// THIS SHOULD BE COPIED AND NOT EXTENDED!!!
FUNCTION_BLOCK ABSTRACT AbstractRoom IMPLEMENTS I_Execute
VAR CONSTANT
	STATE_CAP		: UDINT := 4;
END_VAR
VAR
	_this			: Entity;
	_ctx			: Room_Ctx;
	_room			: RoomInterface(_ctx);
	_tag			: Tag(CONCAT('Room_', UDINT_TO_STRING(_room.Id)));
	_compTag		: Comp(_tag, _this);
	_exe			: Execute(THIS^);
	
	_uiLogic		: Room_UiLogic(_ctx);
	
	_onSystemEvent	: Room_OnSystemEvent(_ctx);
	
	_smgr			: StateManager<STATE_CAP>(_this);
	_proxSmgr		: StateManagerProxy(_smgr, _ctx.state.iMgr);
	
	_disable		: Room_State_Disabled(_this, _ctx);
	_proxDisable	: StateProxy(_disable, _ctx.state.iDisable);
	
	_fault			: Room_State_Fault(_this,_ctx);
	_proxFault		: StateProxy(_fault, _ctx.state.iFault);	
	
	_idle			: Room_State_Idle(_this,_ctx);
	_proxIdle		: StateProxy(_idle, _ctx.state.iIdle);	
	
	_systemOff		: Room_State_SystemOff(_this,_ctx);
	_proxSystemOff	: StateProxy(_systemOff, _ctx.state.iSystemOff);
END_VAR

	// Here add custom components

METHOD Execute
END_METHOD

METHOD Init
_smgr.Request(_idle);
END_METHOD

END_FUNCTION_BLOCK

(* stored: Version 1.1.0.1
   POU AbstractRoom: Id {2e0e75c6-de15-4761-ae40-14041f36bdf4}, SpecialFunc None
   Method Execute: Id {51b956d4-c76f-41de-a458-174fed593c72}
   Method Init: Id {3ff82767-55bc-4f86-a241-d582f5293491} *)
